Universal Robots URScript: test lift column position.script

def test_lift_column_position():
  global _hidden_verificationVariable=0
  set_target_payload(10.450000, [0.000000, -0.064000, 0.064000], [0.076889, 0.076889, 0.076889, 0.000000, 0.000000, 0.000000])
  set_tcp(p[0.00451,-0.328,0.10639,1.2092,-1.2092,1.2092])
  set_standard_analog_input_domain(0, 1)
  set_standard_analog_input_domain(1, 1)
  set_tool_analog_input_domain(0, 1)
  set_tool_analog_input_domain(1, 1)
  set_analog_outputdomain(0, 0)
  set_analog_outputdomain(1, 0)
  set_input_actions_to_default()
  set_tool_communication(False, 115200, 0, 1, 1.5, 3.5)
  set_tool_output_mode(0)
  set_tool_digital_output_mode(0, 1)
  set_tool_digital_output_mode(1, 1)
  set_tool_voltage(0)
  set_gravity([0.0, 0.0, 9.82])
  set_safety_mode_transition_hardness(1)
  global Point_1=p[0.0,0.0,0.0,0.0,0.0,0.0]
  # begin: URCap Installation Node
  #   Source: MachineLogic for Universal Robots, 3.1.7, Vention Inc.
  #   Type: MachineLogic for Universal Robots
  def waitForResponse(expected_response_vention, cname_vention):
  response_vention = socket_read_string(cname_vention,timeout=15)
  while response_vention != expected_response_vention:
  sleep(0.01)
  response_vention = socket_read_string(cname_vention,timeout=15)
  end
  sleep(0.01)
  sync()
  end
  def sendString(string_vention, expected_response_vention, cname_vention):
  socket_send_string(str_cat(string_vention,";"), cname_vention)
  response_vention = socket_read_string(cname_vention,timeout=15)
  if(response_vention == "nAck"):
  popup("nAck received")
  end
  while response_vention != expected_response_vention:
  sleep(0.01)
  response_vention = socket_read_string(cname_vention,timeout=15)
  if(response_vention == "nAck"):
  popup("nAck received")
  end
  end
  sleep(0.01)
  sync()
  end
  def sendStringNAck(string_vention, expected_response_vention, cname_vention):
  socket_send_string(str_cat(string_vention,";"), cname_vention)
  response_vention = socket_read_string(cname_vention,timeout=15)
  if(response_vention == "nAck"):
  popup("nAck received")
  end
  while(response_vention != expected_response_vention and response_vention != "nAck"):
  sleep(0.01)
  response_vention = socket_read_string(cname_vention,timeout=15)
  if(response_vention == "nAck"):
  popup("nAck received",blocking=True)
  end
  end
  sleep(0.01)
  sync()
  end
  def sendStringWithTimeout(string_vention, expected_response_vention, cname_vention):
  socket_send_string(str_cat(string_vention,";"), cname_vention)
  response_vention = socket_read_string(cname_vention,timeout=10)
  if(response_vention == "nAck"):
  popup("nAck received"+string_vention)
  end
  sleep(0.01)
  sync()
  end
  def pollString(string_vention, expected_response_vention, cname_vention):
  socket_send_string(str_cat(string_vention,";"), cname_vention)
  response_vention = socket_read_string(cname_vention,timeout=15)
  if(response_vention == "nAck"):
  popup("nAck received")
  end
  while response_vention != expected_response_vention:
  sleep(1)
  socket_send_string(str_cat(string_vention,";"), cname_vention)
  response_vention = socket_read_string(cname_vention,timeout=15)
  if(response_vention == "nAck"):
  popup("nAck received")
  end
  end
  sleep(0.01)
  sync()
  end
  def sendVariable(var_vention, data_vention, expected_response_vention, cname_vention):
  socket_set_var(var_vention, data_vention, cname_vention)
  response_vention = socket_read_string(cname_vention,timeout=15)
  if(response_vention == "nAck"):
  popup("nAck received")
  end
  while response_vention != expected_response_vention:
  sleep(0.01)
  response_vention = socket_read_string(cname_vention,timeout=15)
  if(response_vention == "nAck"):
  popup("nAck received")
  end
  end
  sleep(0.01)
  sync()
  end
  def intToString(integer_vention,cname_vention):
  stringFix=""
  multiplier_vention123=1
  if integer_vention<0:
  stringFix="-"
  multiplier_vention123=-1
  end
  socket_set_var("GetString",integer_vention*multiplier_vention123,cname_vention)
  string_vention=""
  while string_vention=="":
  sleep(0.01)
  string_vention=socket_read_string(cname_vention,timeout=15)
  end
  sleep(0.01)
  sync()
  string_vention=stringFix+string_vention
  return string_vention
  end
  string_vention=""
  isVentionMovementBusy = False
  isVentionParallelMovementSendingScript = False
  ventionThreadHandle = 1
  isVentionMovementBusyMachineMotion1 = False
  isVentionParallelMovementSendingScriptMachineMotion1 = False
  socket_vention = socket_open("192.168.3.52", 9999, "MachineMotion1")
  if socket_vention==False:
  popup("Check configuration, can't connect to MachineMotion")
  end
  waitForResponse("MachineMotion connection established", "MachineMotion1")
  sendString("isReady", "MachineMotion isReady = true", "MachineMotion1")
  sendStringWithTimeout("setURCapVersion2", "setURCapVersion loaded", "MachineMotion1")
  sendString("SET speed_v2 1000000", "Ack", "MachineMotion1")
  sendString("SET acceleration_v2 100000", "Ack", "MachineMotion1")
  sendString("SET de_axis_1_microsteps_config 8", "Ack", "MachineMotion1")
  sendString("SET de_axis_1_mechanical_gain_config_v2 150000.0", "Ack", "MachineMotion1")
  sendString("SET de_axis_1_direction_config 1", "Ack", "MachineMotion1")
  sendString("SET de_axis_1_type_config Custom Actuator ", "Ack", "MachineMotion1")
  sendString("de_axis_1_config_exec", "Ack", "MachineMotion1")
  # end: URCap Installation Node
  # begin: URCap Installation Node
  #   Source: WireTank Serial, 4.9.0, WireTank, LLC
  #   Type: WireTank Serial
  WTSerialBridge = rpc_factory("xmlrpc","http://127.0.0.1:40511/RPC2")
  # end: URCap Installation Node
  step_count_d95dbc34_0ea6_4a02_a4ff_8c3efa7da4c6 = 0.0
  thread Step_Counter_Thread_da4826b4_98a7_4c5e_bafb_61614a063054():
    while (True):
      step_count_d95dbc34_0ea6_4a02_a4ff_8c3efa7da4c6 = step_count_d95dbc34_0ea6_4a02_a4ff_8c3efa7da4c6 + 1.0
      sync()
    end
  end
  run Step_Counter_Thread_da4826b4_98a7_4c5e_bafb_61614a063054()
  $ 2 "Robot Program"
  $ 3 "'test'"
  # 'test'
  $ 4 "var_1≔0.0"
  global var_1=0.0
  # begin: URCap Program Node
  #   Source: MachineLogic for Universal Robots, 3.1.7, Vention Inc.
  #   Type: MachineLogic for Universal Robots
  $ 5 "MachineLogic Get Position"
  while isVentionMovementBusyMachineMotion1==True:
  sleep(0.05)
  end
  if(isVentionMovementBusyMachineMotion1 == False):
  isVentionMovementBusyMachineMotion1 = True
  socket_send_string("estop/status;", "MachineMotion1")
  temp_estop_var_vention = socket_read_string("MachineMotion1",timeout=15)
  while(temp_estop_var_vention=="estop/status true"):
  if temp_estop_var_vention=="estop/status true":
  sendStringWithTimeout("estop/systemreset/request","Ack estop/systemreset/request;","MachineMotion1")
  end
  socket_send_string("estop/status;", "MachineMotion1")
  temp_estop_var_vention = socket_read_string("MachineMotion1",timeout=15)
  if temp_estop_var_vention=="estop/status true":
  popup("MachineMotion in estop, make sure you have all emergency modules released manually. If you continue the system will try to reset MachineMotion automatically.",blocking=True)
  end
  end
  else:
  popup("resource is being used already: MachineMotion1")
  halt
  end
  socket_send_string("GET im_get_controller_pos_axis_1;", "MachineMotion1")
  temp_drive = socket_read_ascii_float(1, "MachineMotion1",timeout=15)
  global var_1 = temp_drive[1]
  isVentionMovementBusyMachineMotion1 = False
  sleep(0.03)
  # end: URCap Program Node
  $ 6 "Popup"
  popup(str_cat("",var_1), "Message", False, False, blocking=True)
end
